(*
Nazwa:			FB_WeightCorrection
Opis:			Korekcja wagi
Wersja:			v1.3
Data:			2019-11-28
Autor:			TW,DP
Urzadzenia:		Korekta wagi 
Konfiguracja:	
Info: 
-wyłączono wpisywanie maksymalnej korekty bo to bez sensu, ze wpisywało np -15
-poprawiono warningi, które wskazywalo w kompilatorze
-poprawiony blad maksymalnej korekty (minus przerabia na plus)
*)

FUNCTION_BLOCK FB_WeightCorrection
VAR_INPUT
	bEnable:BOOL;					//Zezwolenie na pracę automatycznej korekcji
	bReset:BOOL;					//Reset korekcji dozy i obliczonej gęstości
	bAddMeasurment:BOOL;			//Dodanie pomiaru wagi do rozpatrzenia korekcji dozy
	lrActualDoseVolumeSV:LREAL;		//Aktualna wartość nastawy objetości dozy (ta która jest nastawiona na dozowniku)
	lrDoseVolumeSV:LREAL;			//Wartość nastawy objetości dozy dla danego opakowania (wartość z rejestru)  [ml]
	lrMassWeightSV:LREAL;			//Zadana wartość masy produktu [g]
	lrDoseMeasurment:LREAL;			//Wartość masy odczytana z wagi [g]
	lrDensity:LREAL;				//Gęstość masy g/ml (Jeśli wartość 0, oblicz z wydozowanej ostatniej wartości)
	lrMeasurmentCorrection:LREAL;	//Korekcja wskazania wagi [g]
	lrConteinerWeight:LREAL;			//Waga kubeczka [g]
	lrWholePackWeight:LREAL;		//Waga kubeczka razem z platynką i nakrętką itp. [g]
	lrUpperTolerance:LREAL;			//Górna granica tolerancji
	lrLowerTolerance:LREAL;			//Dolna granica tolerancji	
	nMaxMeasurmentDiff:LREAL;		//Maksymalna różnica pomiędzy pomiarami
	nMaxCorrectionVolume:UDINT;		//Maksymalna nastawa dozy korekcji
	nNrOfMeasurment:UINT;			//Ilość próbek do uśrednienia wartości korekcji dozy
	lrCorrectionStep: LREAL;		//Skok korekcji dozy [ml]
	_ALARMINFO_ :BOOL;
	iStationIndex:UDINT;					//Numer stacji 
	sStationName:STRING;					//Nazwa stacji	

END_VAR
VAR_OUTPUT
	lrMeasuredDensity:LREAL;		//Obliczona wartość gęstości [g/ml]
	lrDoseMaxOdds:LREAL;			//Najwieksze różnice pomiędzy wagami wydozowań
	nMeasurmentCount:UINT;			//Ilość zebranych pomiarów do uśrednienia wagi
	bError:BOOL; 					//Błąd korekcji <=0
	nErrorNr:UDINT;					//Numer Błędu
	sErrorDescription:STRING;		//Opis błędu 
	sErrorDescription2: STRING;				//Opis błędu 2
	sErrorStationName:STRING;				//Nazwa stacji
	udiStationID:UDINT;				// Nr stacji

	lrAverageCounted:LREAL;			//średnia z ostatnich pomiarów
END_VAR
VAR_IN_OUT
	lrDoseVolumeCorrection:LREAL;			//Wartość korekty dozy [ml]
END_VAR
VAR
	rtAddMeasurment: R_TRIG;
	aMeasuredWeight: ARRAY [1..10] OF LREAL;
	
	i: UINT;
	// Suma pomiarów wag
	lrMeasureSum: LREAL;
	// Średnia pomiarów wagi
	lrAverageWeight: LREAL;
	lrUsedDensity:LREAL;
	// trigger Resetu
	rtrigReset: R_TRIG;
	// poprzednia wartość dozy kontrolowanej butelki [ml]
	lrLastDoseVolumeSV: LREAL :=89033008911;
	lrDoseVolumeCorrectionTemp: LREAL;
	Delta: DINT;
	bWeightTooLow:BOOL;
	bWeightTooHigh:BOOL;
	lrWeightHisteresisCenter:LREAL;//
END_VAR

aStationID();
rtAddMeasurment(CLK:=bAddMeasurment,Q=>);


IF bEnable THEN
	
	
	//Jeśli odczytana nowa doza 
	IF rtAddMeasurment.Q THEN
		
		//Jeśli dozy różne zacznij próbkowanie wag od początku
		IF lrActualDoseVolumeSV<>lrDoseVolumeSV THEN
			nMeasurmentCount:=0;
			lrMeasureSum:=0;
		
		//jeśli nastawy zgadzają sie 	
		ELSE	
		
			lrLastDoseVolumeSV:=lrDoseVolumeSV;
			bError:=FALSE;
			nMeasurmentCount:=nMeasurmentCount+1;
			aMeasuredWeight[nMeasurmentCount]:=lrDoseMeasurment-lrConteinerWeight+lrMeasurmentCorrection;
			lrMeasureSum:=lrMeasureSum+aMeasuredWeight[nMeasurmentCount];
			
			IF nMeasurmentCount=1 THEN
				lrDoseMaxOdds:=0;
			END_IF
			
			//Sprawdzanie największych odchyłek w wadze miedzy pomiarami
			FOR i:=1 TO nMeasurmentCount DO
				IF ABS(aMeasuredWeight[i]-aMeasuredWeight[nMeasurmentCount])>lrDoseMaxOdds THEN
					lrDoseMaxOdds:=ABS(aMeasuredWeight[i]-aMeasuredWeight[nMeasurmentCount]);
				END_IF
			END_FOR
			

		END_IF
		
		IF lrDoseMaxOdds>nMaxMeasurmentDiff THEN
				nMeasurmentCount:=0;
				lrMeasureSum:=0;
		END_IF
		//Obliczanie korekty jeśli ilość próbek pomiarowych została osiągnięta
		IF nMeasurmentCount>=(nNrOfMeasurment) THEN
			lrAverageWeight:=lrMeasureSum/UINT_TO_LREAL(nMeasurmentCount);
			lrAverageCounted:=lrAverageWeight;
			lrMeasureSum:=0;
			//lrMeasuredDensity:=(lrAverageWeight)/(lrDoseVolumeSV(*+lrDoseVolumeCorrection*)+0.000000000001);
			IF lrDensity>0 THEN
				lrUsedDensity:=lrDensity;
			ELSE
				//lrUsedDensity:=lrMeasuredDensity;
				bError:=TRUE;
				nErrorNr:=211;
				sErrorDescription:='Zadana wartość gęstości poniżej 0.';
			END_IF
			
			
			//Jeśli nie ma błędu oblicz korektę
			IF NOT bError (*AND (((LREAL_TO_DINT(lrMassWeightSV)-LREAL_TO_DINT(lrAverageWeight))>=ABS(lrLowerTolerance)) OR (((LREAL_TO_DINT(lrAverageWeight)-LREAL_TO_DINT(lrMassWeightSV)>=ABS(lrUpperTolerance)))))*) THEN
				
			
				Delta:=(LREAL_TO_DINT(lrMassWeightSV)-LREAL_TO_DINT(lrAverageCounted));
				
			//	lrWeightHisteresisCenter:=(LREAL_TO_DINT(lrMassWeightSV)+((ABS(lrLowerTolerance)+ABS(lrUpperTolerance))/2)-(ABS(lrLowerTolerance)));
				// 04.11.2022 Dązy do zadanej bez środka
				lrWeightHisteresisCenter:=lrMassWeightSV;
				
				//Wykrywanie czy waga przekracza górny zakres widełek
				IF LREAL_TO_DINT(lrAverageCounted)<LREAL_TO_DINT(lrWeightHisteresisCenter) THEN
					bWeightTooLow:=TRUE;
					bWeightTooHigh:=FALSE;
			   //Wykrywanie czy waga przekracza dolną granicę widełek
				ELSIF LREAL_TO_DINT(lrAverageCounted)>LREAL_TO_DINT(lrWeightHisteresisCenter)THEN
					bWeightTooLow:=FALSE;
					bWeightTooHigh:=TRUE;
				END_IF
				
				
				
				//Jeśli osiągnieta wartość miedzy widełkami wyłącz podnoszenie dozy
				IF LREAL_TO_DINT(lrAverageCounted)>=(LREAL_TO_DINT(lrMassWeightSV)+((ABS(lrLowerTolerance)+ABS(lrUpperTolerance))/2)-(ABS(lrLowerTolerance))) THEN
					bWeightTooLow:=FALSE;
				END_IF
				
				//Jeśli osiągnieta wartość miedzy widełkami wyłącz obniżanie dozy
				IF LREAL_TO_DINT(lrAverageCounted)<=(LREAL_TO_DINT(lrMassWeightSV)+((ABS(lrLowerTolerance)+ABS(lrUpperTolerance))/2)-(ABS(lrLowerTolerance)))THEN
					bWeightTooHigh:=FALSE;
				END_IF
				
				//Zwiększ dozę jeśli za mała wartość
				IF bWeightTooLow THEN
					IF ABS(LREAL_TO_DINT(lrMassWeightSV)-LREAL_TO_DINT(lrAverageCounted))>10 THEN
						;//lrDoseVolumeCorrection:=lrDoseVolumeCorrection+ABS(LREAL_TO_DINT(lrMassWeightSV)-LREAL_TO_DINT(lrAverageCounted));//wyłączone max
					ELSE
						lrDoseVolumeCorrection:=lrDoseVolumeCorrection+lrCorrectionStep;	
					END_IF
						
						lrLastDoseVolumeSV:=lrDoseVolumeSV;
						
				//Zmniejsz dozę jeśli za duża	
				ELSIF bWeightTooHigh THEN
					IF ABS(LREAL_TO_DINT(lrMassWeightSV)-LREAL_TO_DINT(lrAverageCounted))>10 THEN
						;//lrDoseVolumeCorrection:=lrDoseVolumeCorrection-ABS(LREAL_TO_DINT(lrMassWeightSV)-LREAL_TO_DINT(lrAverageCounted));
					ELSE
						lrDoseVolumeCorrection:=lrDoseVolumeCorrection-lrCorrectionStep;	
					END_IF
					
					lrLastDoseVolumeSV:=lrDoseVolumeSV;
				END_IF
				
				//jeśli korekta poza maksymalnym zakresem, przepisz maksymalny zakres
				IF lrDoseVolumeCorrection>nMaxCorrectionVolume THEN					
					lrDoseVolumeCorrection:=nMaxCorrectionVolume;	
				END_IF
				IF lrDoseVolumeCorrection<-UDINT_TO_LREAL(nMaxCorrectionVolume) THEN					
					lrDoseVolumeCorrection:=-UDINT_TO_LREAL(nMaxCorrectionVolume);	
				END_IF
				
			END_IF;
			nMeasurmentCount:=0;
			lrAverageWeight:=0;
		END_IF	
	END_IF

ELSE
	nMeasurmentCount:=0;
	bError:=FALSE;
	lrDoseMaxOdds:=0;
END_IF

rtrigReset(CLK:=bReset,Q=>);

IF rtrigReset.Q (*AND NOT bError *)THEN
	nMeasurmentCount:=0;
	bError:=FALSE;
	lrDoseMaxOdds:=0;
	lrDoseVolumeCorrection:=0;
	lrMeasuredDensity:=0;
	lrMeasureSum:=0;
END_IF

ErrorHandling();

ACTION aStationID:
udiStationID	:=	iStationIndex;
END_ACTION

ACTION ErrorHandling:

IF bReset THEN
	bError:=FALSE;
	nErrorNr:=0;
	sErrorDescription:='';
	lrDoseMaxOdds:=0;
	lrDoseVolumeCorrectionTemp:=0;
END_IF

IF bEnable THEN
	;
	
ELSE
	bError:=FALSE;
	nErrorNr:=0;
	sErrorDescription:='';	
END_IF


(*Przepisywanie nazwy stacji*)
sErrorStationName := sStationName;
END_ACTION

END_FUNCTION_BLOCK

(* stored: Version 1.1.0.1, ProductVersion 3.1.4026.13, FileIdentifier 89adeb5c84c3d9faa91b46991936aff3c1ee07c3, FileSignature 3526edac44412034ab86430b5bdffd5ffd3913640f350aee4eebc904ea93558f42b3b23b0bfd2b8d53dcd65e6e14bf60c461d0f0e255c28ede98f5286a7a737b4db74c2310c35425c718ec356c9ba60698b700368dfadd9cc50b9bbaf73bc2abb7bb44a9211cd87733bb1e55840293cd065f7aa1a81db6bf50163ce1eda10b3d7413279347ea9ea4b48ce7f0d2501230c3d0f99bddd210395e0fb002f5ad220ce49a10aa8f6884c84bdc2c665397cb5c055914b76828dd1d0a2c2100bda2b2bcf49e633da6dd7a6e3c7285d4ce8a09c0e14168f12568c7febf3e826c2ac6dc0664d1a34f53dd58f7166c6df0e74b5df33497cb9a1e35a8cd3ad4a9e1fcd15c2f
   POU FB_WeightCorrection: Id {b9c7cd89-af72-445a-b3f8-2cb3544af2da}, SpecialFunc None
   Action aStationID: Id {152adb07-838f-443a-abf4-74fea1578ab9}
   Action ErrorHandling: Id {8e6703aa-cc17-469f-ae52-dadb248c8862} *)
